// TIA Portal V19 export
DATA_BLOCK "ParametersControl"   // DB113
// stored: MemoryReserve 100
   VAR
      uploadPlcToHmi : Bool;
      uploadPlcToHmiDone : Bool;
      downloadHmiToPlc : Bool;
      downloadHmiToPlcDone : Bool;
   END_VAR
BEGIN
END_DATA_BLOCK
